           //enable of single controller actions
           //----------------------------------- 
           IF ("AC".CTL_AV_SPD_TI > 0.0)   THEN         //i- part
               #int_action_on   :=  true;
           ELSE
               #int_action_on   :=  false;
           END_IF;

           IF ("AC".CTL_AV_SPD_TD > 0.0)   THEN         //d-part
               #der_action_on   :=  true;
           ELSE
               #der_action_on   :=  false;
           END_IF;

           //call Standard PID controller 
           //----------------------------
           #STD_PID(COM_RST         :=  "KYD".SPD_CTRL_RST,                   //restart of controller, resets controller values
                   MAN_ON          :=  NOT #ctl_avg_spd_on,                 //switch controller on/off
                   PVPER_ON        :=  false,                              //activate reading of peripherie value
                   P_SEL           :=  true,                               //proportional action on
                   I_SEL           :=  #int_action_on,                      //integral action on
                   INT_HOLD        :=  #int_hold_req,                       //integral action hold
                   I_ITL_ON        :=  false,                              //initialization of the integral action - set value of I_ITLVAL
                   D_SEL           :=  #der_action_on,                      //derivative action on
                   CYCLE           :=  T#100ms,                            //sample time
                   SP_INT          :=  #set,                                //internal setpoint
                   PV_IN           :=  #act,                                //process variable input
                   PV_PER          :=  W#16#0000,                          //process variable peripherial input
                   MAN             :=  #hand,                               //hand value as percentaged input
                   GAIN            :=  "AC".CTL_AV_SPD_GN,                   //controller gain
                   TI              :=  DINT_TO_TIME(REAL_TO_DINT("AC".CTL_AV_SPD_TI * 1000.0)),  //integration time
                   TD              :=  DINT_TO_TIME(REAL_TO_DINT("AC".CTL_AV_SPD_TD * 1000.0)),  //derivative time
                   TM_LAG          :=  DINT_TO_TIME(REAL_TO_DINT("AC".CTL_AV_SPD_T1 * 1000.0)),  //time lag of the derivative action
                   DEADB_W         :=  0.0,                            //dead band of control deviation
                   LMN_HLM         :=  #hl,                             //upper limit of controller output as percentaged value 
                   LMN_LLM         :=  #ll,                             //lower limit of controller output as percentaged value
                   PV_FAC          :=  1.0,                            //process variable factor (used on peripherial input)
                   PV_OFF          :=  0.0,                            //process variable offset
                   LMN_FAC         :=  1.0,                            //output standardization(percentage to physical value)
                   LMN_OFF         :=  0.0,                            //offset of output value
                   I_ITLVAL        :=  0.0,                            //initialization value of the integral action
                   DISV            :=  #z_input);                       //disturbance variable

                   //write output variables of PID controller
                   //----------------------------------------
                   "CTL".Y_AVG_XT_SPD    :=  #STD_PID.LMN * #ro;               //controller output variable as physical value

                   #per_out         :=  #STD_PID.LMN_PER;    //peripherial controller output variable
                   #high_lim_active :=  #STD_PID.QLMN_HLM;   //high limit of controller output is reached
                   #low_lim_active  :=  #STD_PID.QLMN_LLM;   //low limit of controller output is reached
                   #p_part_out      :=  #STD_PID.LMN_P;      //proportionality component
                   #i_part_out      :=  #STD_PID.LMN_I;      //integral component
                   #d_part_out      :=  #STD_PID.LMN_D;      //derivative component
                   #eff_act_val     :=  #STD_PID.PV;         //effective process variable 
                   #error_sig       :=  #STD_PID.ER;         //control deviation

           //write display values of controller parts
           //----------------------------------------        
           "DIS".AVG_SPD_CONT_P  := #p_part_out * #ro; 
           "DIS".AVG_SPD_CONT_D  := #d_part_out * #ro;
           "DIS".AVG_SPD_CONT_I  := #i_part_out * #ro;

           //evaluate controller output limits
           //---------------------------------
           IF #high_lim_active XOR #low_lim_active   THEN                //check controller limits
               IF (#ctrl_calls > 50) THEN                                   
                   IF #high_lim_active AND (#i_part_out > 0.0)   THEN 
                       #int_hold_req    :=  true;                       //set integral action on hold
                   ELSIF #low_lim_active AND (#i_part_out < 0.0) THEN 
                       #int_hold_req    :=  true;                       //set integral action on hold
                   ELSE 
                       #int_hold_req    :=  false;                      //reset integral action on hold
                   END_IF;
               ELSE
                   #ctrl_calls  :=  #ctrl_calls + 1;                     //count controller calls
               END_IF;
           ELSE
               #ctrl_calls      :=  0;                                  //reset controller call counts
               #int_hold_req    :=  false;                              //reset integral action hold request
           END_IF;

           //switch on average pull speed controller
           //--------------------------------------- 
           IF "SY".CTL_AVG_SPD_ON    THEN 
               #ctl_avg_spd_on  :=  true;
           END_IF;


       //write average speed controller output as setpoint for crucible rotation
       //-----------------------------------------------------------------------    
       IF ("APC".STATUS = "APC".SHOULDER) AND ("PAR_MAIN".SH_CRUC_ROT_CTL_ON = 1.0) THEN
           "CTL".SET_CR_ROT  :=  "CTL".Y_GRW_RTE;
       ELSIF ("APC".STATUS = "APC".BODY) AND ("PAR_MAIN".BY_CRUC_ROT_CTL_ON = 1.0) THEN    
           "CTL".SET_CR_ROT  :=  "CTL".Y_AVG_XT_SPD;
       END_IF;         

       //save actual values for next cycle
       //---------------------------------               
       #z_input_old             :=  #z_input;
       #set_avg_cruc_rot_old    :=  "AC".SET_AVG_CRUC_ROT;
END_FUNCTION_BLOCK

FUNCTION_BLOCK "CM_LOOP_MLT_TMP"   // FB139, SCL
{ S7_Optimized_Access := 'FALSE' }
VERSION : 0.0
// --------------------------------------------------------------------------------
//     program     :    CM_LOOP_MLT_TMP
//     description :    melt temperature control loop 
//     name        :    K. Kalkowski
//     date        :    10.12.99 
// 
//     revision    :    call of CONT_C added as alternative
//     name        :    G. Eibelsh鋟ser
//     date        :    07.09.2007
//     
//     revision    :    
//     name        :    
//     date        :    
// 
//                     (c)PVA TePla AG
//     --------------------------------------------------------------------------------
   VAR
      STD_PID : CONT_C;   // standard Siemens controller algorithm
      PT1 : "CM_PT1";   // pt1 filter for melt temp
      ramp_enb : Bool;
      cyc_cnt : Bool;
      int_hold_req : Bool;   // integral hold action request
      pyr_failed : Bool;
      ctl_mlt_tmp_on : Bool;
      ctrl_calls : Int;   // controller call counter
      i : Int;
      set : Real;   // internal set point
      act : Real;   // internal actual value
      set_ramp : Real;
      pyr_act_melt_tmp_prv : Real;
      set_prv_cyc : Real;
   END_VAR
   VAR_TEMP
      high_lim_active : Bool;   // high limit of controller output is reached
      low_lim_active : Bool;   // low limit of controller output is reached
      int_action_on : Bool;   // integral action on
      der_action_on : Bool;   // derivative action on
      per_out : Word;   // peripherial controller output variable
      p_part_out : Real;   // proportionality component
      i_part_out : Real;   // integral component
      d_part_out : Real;   // derivative component
      eff_act_val : Real;   // effective process variable
      error_sig : Real;   // control deviation
   END_VAR
   VAR CONSTANT
      nc : Real := 0.0;   // "not connected" input
   END_VAR
BEGIN

       //read setpoint from recipe
       //-------------------------                                                
       #set := "AC".SET_MLT_1_TMP;              

       //read filter time from recipe
       //----------------------------
       "AC".CTL_MLT_TMP_1_TF := "PAR_SUB".FI_MLT_TMP_1;

       //call filter algorithm
       //---------------------                                                  
       #PT1 (u_in      := "PAI".PYR_ACT_MELT_TMP,                   
            t1_in     := "AC".CTL_MLT_TMP_1_TF, 
            ts_in     := 0.1,
            tc_in     := 0.1,
            range_in  := "CNF".MLT_TMP_1_RANGE_HI,
            range_out := "CNF".MLT_TMP_1_RANGE_HI,
            y_llim    := "CNF".MLT_TMP_1_RANGE_LOW,
            y_hlim    := "CNF".MLT_TMP_1_RANGE_HI,
            y_out     := "CTL".AVG_MLT_1_TMP);

       "CTL".AVG_MLT_1_TMP   := "CTL".AVG_MLT_1_TMP + "PAR_MAIN".MCONST_MLT_TMP_OFFS;  //add offset to filtered value                          

       #act                 := "CTL".AVG_MLT_1_TMP;
       (*
       //check pyrometer signal when temperature control is on
       //-----------------------------------------------------
       IF SY.CTL_MLT_TMP_ON  THEN
           //calculate deviation of temperature from last cycle
           //--------------------------------------------------
           IF ((pyr_act_melt_tmp_prv - PAI.PYR_ACT_MELT_TMP) > 15.0) THEN  //temp. drop larger 15癈
               pyr_failed  :=  true;
           END_IF;

       ELSE
           //reset signal "pyrometer failed" with delay
           //------------------------------------------
           IF pyr_failed   THEN 
               IF (i > 50)    THEN             //delay reset at least 5 seconds
                   IF NOT APC.AUTOMATIC THEN
                       pyr_failed  :=  false;  //reset failure flag when automatic is off
                   END_IF;
               ELSE 
                   i   :=  i + 1;  //increment 100ms counter
               END_IF; 
           ELSE 
               i   :=  0;  //reset counter value
           END_IF;

       END_IF; 

       //store actual temperature for one 100ms cycle
       //--------------------------------------------
       pyr_act_melt_tmp_prv   :=  PAI.PYR_ACT_MELT_TMP;    

       //set fault message when pyrometer failed
       //---------------------------------------
       FLT.MLT_TMP_SIG   :=  pyr_failed;
       *)
       //built control on flag
       //---------------------                                                    
       IF "APC".AUTOMATIC AND NOT #pyr_failed THEN                         
           "SY".CTL_MLT_TMP_ON := "DC".CTL_MLT_1_TMP_ON;                 
       ELSE 
           "SY".CTL_MLT_TMP_ON := FALSE; 
       END_IF;

       "LT".CTL_MELT_TMP_1_ON := "SY".CTL_MLT_TMP_ON; 

       //melt temperature controller setpoint ramp
       //-----------------------------------------
       IF "SY".CTL_MLT_TMP_ON  THEN

           IF (#set <> #set_prv_cyc) THEN    //compare setpoint with setpoint of previous cycle
               #ramp_enb := true;           //enable ramp when setpoint has changed
           END_IF;
           #set_prv_cyc :=  #set;        //store setpoint of current cycle

           // call setpoint ramp function after controller start
           //---------------------------------------------------
           IF ("PAR_SUB".MELT_TMP_RP_GRAD > 0.0)     THEN
               "CM_SET_RAMP"(rp_enb      := #ramp_enb,
                           i           := #cyc_cnt,
                           max_dev     := "PAR_SUB".MELT_TMP_RP_MAX_DEV,
                           rp_start    := "PAR_SUB".MELT_TMP_RP_START,
                           rp_grad     := "PAR_SUB".MELT_TMP_RP_GRAD,
                           tme_base    := 60.0,
                           tc_in       := 0.1,
                           set_p       := #set,
                           act_v       := #act,
                           set_out     := #set_ramp);

               #set     := #set_ramp; 
           END_IF;
       ELSE
           #ramp_enb  := true;     
           #cyc_cnt   := true;                
       END_IF;

       //set display variables of melt temperature
       //-----------------------------------------
       "DIS".SET_MLT_TMP_1   := #set;
       "DIS".ACT_MLT_TMP_1   := #act;

       //do controller call
       //------------------ 

           //switch off melt temperature controller
           //-------------------------------------- 
           IF NOT "SY".CTL_MLT_TMP_ON   THEN 
               #ctl_mlt_tmp_on  :=  false;
           END_IF;

           //enable of single controller actions
           //----------------------------------- 
           IF ("AC".CTL_MLT_TMP_1_TI > 0.0)   THEN         //i- part
               #int_action_on   :=  true;
           ELSE
               #int_action_on   :=  false;
           END_IF;

           IF ("AC".CTL_MLT_TMP_1_TD > 0.0)   THEN         //d-part
               #der_action_on   :=  true;
           ELSE
               #der_action_on   :=  false;
           END_IF;

           //call Standard PID controller 
           //----------------------------
           #STD_PID(COM_RST         :=  "KYD".MLT_TMP_CTRL_RST,               //restart of controller, resets controller values
                   MAN_ON          :=  NOT #ctl_mlt_tmp_on,                 //switch controller on/off
                   PVPER_ON        :=  false,                              //activate reading of peripherie value
                   P_SEL           :=  true,                               //proportional action on
                   I_SEL           :=  #int_action_on,                      //integral action on
                   INT_HOLD        :=  #int_hold_req,                       //integral action hold
                   I_ITL_ON        :=  false,                              //initialization of the integral action - set value of I_ITLVAL
                   D_SEL           :=  #der_action_on,                      //derivative action on
                   CYCLE           :=  T#100ms,                            //sample time
                   SP_INT          :=  #set,                                //internal setpoint
                   PV_IN           :=  #act,                                //process variable input
                   PV_PER          :=  W#16#0000,                          //process variable peripherial input
                   MAN             :=  0.0,                                //hand value as percentaged input
                   GAIN            :=  "AC".CTL_MLT_TMP_1_GN,                //controller gain
                   TI              :=  DINT_TO_TIME(REAL_TO_DINT("AC".CTL_MLT_TMP_1_TI * 1000.0)), //integration time
                   TD              :=  DINT_TO_TIME(REAL_TO_DINT("AC".CTL_MLT_TMP_1_TD * 1000.0)), //derivative time
                   TM_LAG          :=  DINT_TO_TIME(REAL_TO_DINT("AC".CTL_MLT_TMP_1_T1 * 1000.0)), //time lag of the derivative action
                   DEADB_W         :=  0.0,                            //dead band of control deviation
                   LMN_HLM         :=  100.0,                          //upper limit of controller output as percentaged value 
                   LMN_LLM         :=  -100.0,                         //lower limit of controller output as percentaged value
                   PV_FAC          :=  1.0,                            //process variable factor (used on peripherial input)
                   PV_OFF          :=  0.0,                            //process variable offset
                   LMN_FAC         :=  1.0,                            //output standardization(percentage to physical value)
                   LMN_OFF         :=  0.0,                            //offset of output value
                   I_ITLVAL        :=  0.0,                            //initialization value of the integral action
                   DISV            :=  #nc);                            //disturbance variable

                   //write output variables of PID controller
                   //----------------------------------------
                   "CTL".Y_MLT_1_TMP :=  #STD_PID.LMN / 100.0 * "CNF".HTR_1_TMP_RANGE_HI;   //controller output variable as physical value

                   #per_out         :=  #STD_PID.LMN_PER;                    //peripherial controller output variable
                   #high_lim_active :=  #STD_PID.QLMN_HLM;                   //high limit of controller output is reached
                   #low_lim_active  :=  #STD_PID.QLMN_LLM;                   //low limit of controller output is reached
                   #p_part_out      :=  #STD_PID.LMN_P;                      //proportionality component
                   #i_part_out      :=  #STD_PID.LMN_I;                      //integral component
                   #d_part_out      :=  #STD_PID.LMN_D;                      //derivative component
                   #eff_act_val     :=  #STD_PID.PV;                         //effective process variable 
                   #error_sig       :=  #STD_PID.ER;                         //control deviation

           //evaluate controller output limits
           //---------------------------------
           IF #high_lim_active XOR #low_lim_active   THEN                //check controller limits
               IF (#ctrl_calls > 50) THEN                                   
                   IF #high_lim_active AND (#i_part_out > 0.0)   THEN 
                       #int_hold_req    :=  true;                       //set integral action on hold
                   ELSIF #low_lim_active AND (#i_part_out < 0.0) THEN 
                       #int_hold_req    :=  true;                       //set integral action on hold
                   ELSE 
                       #int_hold_req    :=  false;                      //reset integral action on hold
                   END_IF;
               ELSE
                   #ctrl_calls  :=  #ctrl_calls + 1;                     //count controller calls
               END_IF;
           ELSE
               #ctrl_calls      :=  0;                                  //reset controller call counts
               #int_hold_req    :=  false;                              //reset integral action hold request
           END_IF;

           //switch on melt temperature controller
           //------------------------------------- 
           IF "SY".CTL_MLT_TMP_ON   THEN 
               #ctl_mlt_tmp_on  :=  true;
           END_IF;
END_FUNCTION_BLOCK

FUNCTION_BLOCK "CM_LOOP_GRW_RTE"   // FB140, SCL
{ S7_Optimized_Access := 'FALSE' }
VERSION : 0.0
// --------------------------------------------------------------------------------
//     program     :    CM_LOOP_GRW_RTE
//     description :    growth rate control loop 
//     name        :    K. Kalkowski
//     date        :    12.12.99
// 
//     revision    :    call of CONT_C added as alternative
//     name        :    G. Eibelsh鋟ser
//     date        :    07.09.2007
//     
//     revision    :    
//     name        :    
//     date        :    
// 
//                     (c)PVA TePla AG
//     --------------------------------------------------------------------------------
   VAR
      STD_PID : CONT_C;   // standard Siemens controller algorithm
      DT1 : "CM_DT1";   // dt1 filter for act gtrowth rate
      ramp_enb : Bool;
      cyc_cnt : Bool;
      int_hold_req : Bool;   // integral hold action request
      ctl_grw_rte_on : Bool;
      ctrl_calls : Int;   // controller call counter
      set : Real;   // internal set point
      act : Real;   // internal actual value
      hand : Real;   // internal hand value
      ll : Real;   // controller output low limit
      hl : Real;   // controller output high limit
      ro : Real;   // controller output range
      set_ramp : Real;
      z_input : Real;   // interference input
      z_input_old : Real;   // interference input of previous cycle
      set_avg_cruc_rot_old : Real;   // average crucible rotation setpoint of previous cycle
   END_VAR
   VAR_TEMP
      high_lim_active : Bool;   // high limit of controller output is reached
      low_lim_active : Bool;   // low limit of controller output is reached
      int_action_on : Bool;   // integral action on
      der_action_on : Bool;   // derivative action on
      per_out : Word;   // peripherial controller output variable
      p_part_out : Real;   // proportionality component
      i_part_out : Real;   // integral component
      d_part_out : Real;   // derivative component
      eff_act_val : Real;   // effective process variable
      error_sig : Real;   // control deviation
      act_tmp : Real;   // internal actual value
   END_VAR
   VAR CONSTANT
      nc : Real := 0.0;   // "not connected" input
   END_VAR
BEGIN


       IF "PAR_MAIN".SH_CRUC_ROT_CTL_ON = 1.0 THEN
           IF   ("APC".STATUS = "APC".SHOULDER)   THEN

               IF  "APC".AUTOMATIC  AND NOT "SY".CTL_CR_ROT_SMI    THEN  
                   IF  "DV".START_SH_FLAG     THEN
                       #hand    :=  "PAR_MAIN".SH_START_CRUC_ROT; //crucible rotation setpoint provided from main page
                   ELSIF "DV".TRANS_SH_BY_FLAG  THEN
                       #hand    := "CTL".SET_CR_ROT;              //keep last controller setpoint as setpoint for transistion    
                   END_IF;           
               ELSE
                   #hand := "CM_INSELECT" (auto  := ("APC".AUTOMATIC AND NOT "SY".CTL_CR_ROT_SMI),        
                                       track  := false,
                                       ac     := "AC".SET_CR_ROT,                
                                       kya    := "KYA".SET_CR_ROT);
               END_IF;

               //transform to percentage value
               //-----------------------------
               IF "DV".GRW_RTE_CTRL_STD_ALG  THEN    //only when standard PID algorithm is active
                   #hand    :=  #hand / "CNF".CR_ROT_RANGE * 100.0;
               END_IF;

           END_IF;
       ELSE
           #hand := 0.0;
       END_IF;   

       //read setpoint from recipe
       //-------------------------                              
       #set := "AC".SET_GRW_RTE;         

       //read filter time from recipe
       //----------------------------
       "AC".CTL_GRO_TF := "PAR_SUB".FI_GRO_SH;                

       //call derivative algorithm
       //-------------------------
       #DT1 (u_in       := "AV".ACT_XT_DIA * 600,                   //build actual value   
            td_in      := 0.10,                //mm/min                                
            t1_in      := "AC".CTL_GRO_TF, 
            ts_in      := 1.0,
            tc_in      := 0.1,
            range_in   := "CNF".XT_LFT_RANGE,  
            range_out  := "CNF".XT_LFT_RANGE,
            y_llim     := ("CNF".XT_LFT_RANGE * (-1)),
            y_hlim     := "CNF".XT_LFT_RANGE,
            y_out      := "CTL".ACT_GRW_RTE);

       "DIS".ACT_XTAL_GRO := "CTL".ACT_GRW_RTE;
       #act              := "CTL".ACT_GRW_RTE;                 

       //build control on flag
       //---------------------
       IF "APC".AUTOMATIC THEN                               
           IF "SY".CTL_AVG_CRUC_ROT_ON   THEN
               IF  NOT "SY".CTL_CR_ROT_SMI   THEN
                   "SY".CTL_GRW_RTE_ON := "DC".CTL_GRW_RTE_ON; //set flag according to process mode                 
               ELSE 
                   "SY".CTL_GRW_RTE_ON := FALSE;             //switch off if cruc rot is in semi mode
               END_IF;
           ELSE    
               IF NOT "SY".CTL_HTR_1_SMI THEN 
                   "SY".CTL_GRW_RTE_ON := "DC".CTL_GRW_RTE_ON; //set flag according to process mode
               ELSE
                   "SY".CTL_GRW_RTE_ON := FALSE;
               END_IF;        
           END_IF;
       ELSE
           "SY".CTL_GRW_RTE_ON := FALSE;                     //switch off growth rate control in manuell mode
       END_IF;        

       "LT".CTL_GRO_ON := "SY".CTL_GRW_RTE_ON;                 //set light variable for growth control on         

       //check controller output range
       //-----------------------------
       IF ("APC".STATUS = "APC".SHOULDER)  AND ("PAR_MAIN".SH_CRUC_ROT_CTL_ON = 1.0)  THEN

           IF "SY".CTL_GRW_RTE_ON    THEN
               IF "DV".GRW_RTE_CTRL_STD_ALG  THEN 
                   #ll  :=  "AC".SET_CRUC_ROT_DEV_2 / "CNF".CR_ROT_RANGE * 100.0;
                   #hl  :=  "AC".SET_CRUC_ROT_DEV_1 / "CNF".CR_ROT_RANGE * 100.0;
                   #ro  :=  "CNF".CR_ROT_RANGE / 100.0;
               ELSE
                   #ll  :=  "AC".SET_CRUC_ROT_DEV_2;
                   #hl  :=  "AC".SET_CRUC_ROT_DEV_1;
                   #ro  :=  "CNF".CR_ROT_RANGE;
               END_IF;

           ELSE
               IF "DV".GRW_RTE_CTRL_STD_ALG  THEN 
                   #ll  :=  0.0;
                   #hl  :=  100.0;
                   #ro  :=  "CNF".CR_ROT_RANGE / 100.0;
               ELSE
                   #ll  :=  0.0;
                   #hl  :=  "CNF".CR_ROT_RANGE;
                   #ro  :=  "CNF".CR_ROT_RANGE;
               END_IF;
           END_IF;      
       ELSE
           IF "DV".GRW_RTE_CTRL_STD_ALG  THEN 
               #ll  :=  -100.0;
               #hl  :=  100.0;
               #ro  :=  "CNF".HTR_1_TMP_RANGE_HI / 100.0;
           ELSE
               #ll  :=  "CNF".HTR_1_TMP_RANGE_HI *(-1);
               #hl  :=  "CNF".HTR_1_TMP_RANGE_HI;
               #ro  :=  "CNF".HTR_1_TMP_RANGE_HI;
           END_IF;
       END_IF;

       IF "SY".CTL_GRW_RTE_ON  THEN
           // call setpoint ramp function after controller start
           //---------------------------------------------------
           IF ("PAR_SUB".GRO_RP_GRAD > 0.0)     THEN
               IF #act < 0.0    THEN
                   #act_tmp := 0.0;     //set act_tmp to zero if act < zero
               ELSE
                   #act_tmp := #act;        
               END_IF;    

               "CM_SET_RAMP"(rp_enb      := #ramp_enb,
                           i           := #cyc_cnt,
                           max_dev     := "PAR_SUB".GRO_RP_MAX_DEV,
                           rp_start    := "PAR_SUB".GRO_RP_START,
                           rp_grad     := "PAR_SUB".GRO_RP_GRAD,
                           tme_base    := 60.0,
                           tc_in       := 0.1,
                           set_p       := #set,
                           act_v       := #act_tmp,
                           set_out     := #set_ramp);

               #set     := #set_ramp; 
           END_IF;
       ELSE
           #ramp_enb  := TRUE;     
           #cyc_cnt   := TRUE;                
       END_IF;
       //write display value with setpoint
       //---------------------------------
       "DIS".SET_XTAL_GRO := #set;

       //reset saved interference variables for cruc rot control if growth rate controller is off
       //----------------------------------------------------------------------------------------
       IF   "SY".CTL_GRW_RTE_ON =   FALSE    THEN
           #z_input_old          := 0.0;
           #set_avg_cruc_rot_old := "AC".SET_AVG_CRUC_ROT;
       END_IF;                            

       //change polarity of setpoint and actual if crucible rotation control is off
       //--------------------------------------------------------------------------
       IF ("PAR_MAIN".SH_CRUC_ROT_CTL_ON = 0.0) THEN
           #set     := #set *(-1);
           #act     := #act *(-1);
           #z_input := 0.0;             // keep interference input 0.0, if crucible rotation control is off

       //set interference input with average crucible rotation profile
       //-----------------------------------------------------------------    
       ELSE
           #z_input := #z_input_old + (#set_avg_cruc_rot_old - "AC".SET_AVG_CRUC_ROT) * (-1);   

           //transform to percentage value when standard algorithm is set
           //------------------------------------------------------------
           IF "DV".GRW_RTE_CTRL_STD_ALG  THEN
               #z_input := #z_input / "CNF".CR_ROT_RANGE * 100.0;
           END_IF;
       END_IF;        

       //do controller call
       //------------------

           //switch off growth rate controller
           //---------------------------------
           IF NOT "SY".CTL_GRW_RTE_ON   THEN 
               #ctl_grw_rte_on  :=  false;
           END_IF;

           //enable of single controller actions
           //----------------------------------- 
           IF ("AC".CTL_GRO_TI > 0.0)   THEN             //i- part
               #int_action_on   :=  true;
           ELSE
               #int_action_on   :=  false;
           END_IF;

           IF ("AC".CTL_GRO_TD > 0.0)   THEN             //d-part
               #der_action_on   :=  true;
           ELSE
               #der_action_on   :=  false;
           END_IF;

           //call Standard PID controller 
           //----------------------------
           #STD_PID(COM_RST         :=  "KYD".GRW_RTE_CTRL_RST,               //restart of controller, resets controller values
                   MAN_ON          :=  NOT #ctl_grw_rte_on,                //switch controller on/off
                   PVPER_ON        :=  false,                              //activate reading of peripherie value
                   P_SEL           :=  true,                               //proportional action on
                   I_SEL           :=  #int_action_on,                      //integral action on
                   INT_HOLD        :=  #int_hold_req,                       //integral action hold
                   I_ITL_ON        :=  false,                              //initialization of the integral action - set value of I_ITLVAL
                   D_SEL           :=  #der_action_on,                      //derivative action on
                   CYCLE           :=  T#100ms,                            //sample time
                   SP_INT          :=  #set,                                //internal setpoint
                   PV_IN           :=  #act,                                //process variable input
                   PV_PER          :=  W#16#0000,                          //process variable peripherial input
                   MAN             :=  #hand,                               //hand value as percentaged input
                   GAIN            :=  "AC".CTL_GRO_GN,                      //controller gain
                   TI              :=  DINT_TO_TIME(REAL_TO_DINT("AC".CTL_GRO_TI * 1000.0)), //integration time
                   TD              :=  DINT_TO_TIME(REAL_TO_DINT("AC".CTL_GRO_TD * 1000.0)), //derivative time
                   TM_LAG          :=  DINT_TO_TIME(REAL_TO_DINT("AC".CTL_GRO_T1 * 1000.0)), //time lag of the derivative action
                   DEADB_W         :=  0.0,                            //dead band of control deviation
                   LMN_HLM         :=  #hl,                             //upper limit of controller output as percentaged value 
                   LMN_LLM         :=  #ll,                             //lower limit of controller output as percentaged value
                   PV_FAC          :=  1.0,                            //process variable factor (used on peripherial input)
                   PV_OFF          :=  0.0,                            //process variable offset
                   LMN_FAC         :=  1.0,                            //output standardization(percentage to physical value)
                   LMN_OFF         :=  0.0,                            //offset of output value
                   I_ITLVAL        :=  0.0,                            //initialization value of the integral action
                   DISV            :=  #z_input);                       //disturbance variable

                   //write output variables of PID controller
                   //----------------------------------------
                   "CTL".Y_GRW_RTE   :=  #STD_PID.LMN * #ro;                   //controller output variable as physical value

                   #per_out         :=  #STD_PID.LMN_PER;                    //peripherial controller output variable
                   #high_lim_active :=  #STD_PID.QLMN_HLM;                   //high limit of controller output is reached
                   #low_lim_active  :=  #STD_PID.QLMN_LLM;                   //low limit of controller output is reached
                   #p_part_out      :=  #STD_PID.LMN_P;                      //proportionality component
                   #i_part_out      :=  #STD_PID.LMN_I;                      //integral component
                   #d_part_out      :=  #STD_PID.LMN_D;                      //derivative component
                   #eff_act_val     :=  #STD_PID.PV;                         //effective process variable 
                   #error_sig       :=  #STD_PID.ER;                         //control deviation

           //write display values of controller parts
           //----------------------------------------        
           "DIS".GRW_RTE_CONT_P:= #p_part_out * #ro; 
           "DIS".GRW_RTE_CONT_I:= #i_part_out * #ro;
           "DIS".GRW_RTE_CONT_D:= #d_part_out * #ro;

           //evaluate controller output limits
           //---------------------------------
           IF #high_lim_active XOR #low_lim_active   THEN                //check controller limits
               IF (#ctrl_calls > 50) THEN                                   
                   IF #high_lim_active AND (#i_part_out > 0.0)   THEN 
                       #int_hold_req    :=  true;                       //set integral action on hold
                   ELSIF #low_lim_active AND (#i_part_out < 0.0) THEN 
                       #int_hold_req    :=  true;                       //set integral action on hold
                   ELSE 
                       #int_hold_req    :=  false;                      //reset integral action on hold
                   END_IF;
               ELSE
                   #ctrl_calls  :=  #ctrl_calls + 1;                     //count controller calls
               END_IF;
           ELSE
               #ctrl_calls      :=  0;                                  //reset controller call counts
               #int_hold_req    :=  false;                              //reset integral action hold request
           END_IF;

           //switch on growth rate controller
           //--------------------------------
           IF "SY".CTL_GRW_RTE_ON   THEN 
               #ctl_grw_rte_on  :=  true;
           END_IF;

       //save actual values for next cycle
       //---------------------------------               
       #z_input_old             :=  #z_input;
       #set_avg_cruc_rot_old    :=  "AC".SET_AVG_CRUC_ROT;
END_FUNCTION_BLOCK

FUNCTION_BLOCK "CM_LOOP_MLT_LVL"   // FB141, SCL
{ S7_Optimized_Access := 'FALSE' }
VERSION : 0.0
// --------------------------------------------------------------------------------
//     program     :    CM_LOOP_MLT_LVL
//     description :    melt level control loop 
//     name        :    K. Kalkowski
//     date        :    08.12.99 
// 
//     revision    :    
//     name        :    
//     date        :    
// 
//                     (c)PVA TePla AG
//     --------------------------------------------------------------------------------
   VAR
      P : "CM_P";   // p controller melt level
      PT1 : "CM_PT1";   // pt1 filter for melt level
      ramp_enb : Bool;
      cyc_cnt : Bool;
      enb_mlt_lvl_sft : Bool;
      set : Real;   // internal set point
      act : Real;   // internal actual value
      hand : Real;   // internal hand value
      set_ramp : Real;
      set_cr_spd_cof : Real;
      mlt_lvl_sft_dur : Real;
      act_mlt_lvl_sft : Real;
      mlt_lvl_sft_len : Real;
      mlt_lvl_sft_str_len : Real;
      mlt_lvl_sft_offs_spd : Real;
   END_VAR
   VAR CONSTANT
      nc : Real := 0.0;   // "not connected" input
      min_cr_spd : Real := 0.001;   // [mm/min]
      min_lvl_sft_len : Real := 0.1;   // [mm]
      safety_gap : Real := 5.0;   // safety gap melt level - funnel in [mm]
   END_VAR
BEGIN

       //build hand value 
       //----------------
       IF ("CTL".SET_SPEED_OFFS = 0.0) THEN  //offset speed controller off and output ramped down to zero 
           #hand := "CM_INSELECT" (auto   := ("APC".AUTOMATIC AND NOT "SY".CTL_MLT_LVL_SMI),  //hand value used when melt level controller is off       
                                track  := false,
                                ac     := "AC".SET_CR_SPD,                
                                kya    := "KYA".SET_CR_SPD);  
       ELSE
           #hand := "CTL".SET_CR_SPD; //keep melt level controller output as hand value as long as output of offset speed controller is ramp down to zero
       END_IF;

      //crucible speed coeffizient while tracing of pulling speed is active
      //------------------------------------------------------------------- 
      #set_cr_spd_cof := "CM_INSELECT"   (auto   := ("APC".AUTOMATIC AND NOT "SY".CTL_CR_SPD_COF_SMI),        
                                       track  := true,
                                       ac     := "AC".SET_CR_SPD_COF,                
                                       kya    := "KYA".SET_CR_SPD_COF);                      

       //read filter time from recipe
       //----------------------------
       "AC".CTL_MLT_LVL_TF := "PAR_SUB".FI_MLT_LVL;    

       //built control on flag
       //----------------------
       IF "APC".AUTOMATIC AND NOT "SY".CTL_MLT_LVL_SMI THEN
           "SY".CTL_MLT_LVL_ON := "DC".CTL_MLT_LVL_ON;                 
       ELSE 
           "SY".CTL_MLT_LVL_ON := FALSE; 
       END_IF;

       IF "SY".CTL_MLT_LVL_ON  THEN
           // call setpoint ramp function after controller start
           //---------------------------------------------------
           IF ("PAR_SUB".MLT_LVL_RP_GRAD > 0.0)     THEN

               "CM_SET_RAMP"(rp_enb      := #ramp_enb,
                           i           := #cyc_cnt,
                           max_dev     := "PAR_SUB".MLT_LVL_RP_MAX_DEV,
                           rp_start    := "PAR_SUB".MLT_LVL_RP_START,
                           rp_grad     := "PAR_SUB".MLT_LVL_RP_GRAD,
                           tme_base    := 60.0,
                           tc_in       := 0.1,
                           set_p       := #set,
                           act_v       := #act,
                           set_out     := #set_ramp);

               #set     := #set_ramp; 
           END_IF;
       ELSE
           #ramp_enb  := TRUE;     
           #cyc_cnt   := TRUE;                
       END_IF;


       "LT".CTL_LVL_ON := "SY".CTL_MLT_LVL_ON;                             

       //call P controller
       //-----------------
       #P (set_in        := #set,                        
          act_in        := #act,                
          z_in          := "AV".CRUC_RATIO * "CTL".AVG_XT_SPD * ((#set_cr_spd_cof + "CTL".SET_CR_SPD_COF_OFFS) / 100.0),               
          p_in          := "AC".CTL_MLT_LVL_GN,             
          ts_in         := 0.1,                
          tc_in         := 0.1,            
          tw_in         := 0.5,                
          hand_in       := #hand,            
          range_in      := "CNF".LSR_LVL_RANGE,           //100,               
          range_out     := "CNF".CR_LFT_RANGE,             
          y_llim        := 0.0,                         //(CNF.CR_LFT_RANGE *(-1)),              
          y_hlim        := "CNF".CR_LFT_RANGE,         
          ctrl_on       := "SY".CTL_MLT_LVL_ON,               
          hand_lim_dis  := ("APC".AUTOMATIC AND "DC".CR_LFT_FST),              
          y_out         := "CTL".SET_CR_SPD);         

       //write display value
       //-------------------
       "DIS".SET_CR_SPD_COF  :=  #set_cr_spd_cof;     //write recipe value of crucible speed coefficient to display value

       //set enable flag for melt level shift
       //------------------------------------
       IF ("APC".STATUS = "APC".BODY) THEN
          #mlt_lvl_sft_len       := "PAR_MAIN".BY_MLT_LVL_SFT_LEN;
          #mlt_lvl_sft_str_len   := "PAR_MAIN".BY_MLT_LVL_SFT_STR_LEN;
          #mlt_lvl_sft_offs_spd  := "PAR_MAIN".BY_MLT_LVL_SFT_OFFS_SPD;
       ELSE
          #mlt_lvl_sft_len       := "PAR_MAIN".SH_MLT_LVL_SFT_LEN;
          #mlt_lvl_sft_str_len   := "PAR_MAIN".SH_MLT_LVL_SFT_STR_LEN;
          #mlt_lvl_sft_offs_spd  := "PAR_MAIN".SH_MLT_LVL_SFT_OFFS_SPD;
       END_IF;    

       IF ((ABS(#mlt_lvl_sft_len) < #min_lvl_sft_len) OR (#mlt_lvl_sft_offs_spd < #min_cr_spd)) THEN
           #enb_mlt_lvl_sft     :=  false;
           "FLT".SH_MLT_LVL_SFT  :=  FALSE;
       //negative melt level shift length means lift up of melt level and reduction of melt gap
       //--------------------------------------------------------------------------------------
       ELSIF (("PAR_MAIN".ME_GAP_MLT_FNL > #safety_gap) AND ((#mlt_lvl_sft_len * (-1)) < ("PAR_MAIN".ME_GAP_MLT_FNL - #safety_gap))) THEN 
           #enb_mlt_lvl_sft     :=  true;
           "FLT".SH_MLT_LVL_SFT  :=  FALSE;
       ELSE
           #enb_mlt_lvl_sft :=  false;
           IF ("STA".ACT_STATE = "APC".STATE_RUN) THEN
               "FLT".SH_MLT_LVL_SFT  :=  TRUE;
           ELSE
               "FLT".SH_MLT_LVL_SFT  :=  FALSE;
           END_IF;
       END_IF;

       //melt level shift offset speed calculation in shoulder phase
       //-----------------------------------------------------------
       IF (("APC".STATUS = "APC".BODY) AND "DC".CTL_DIA_ON) OR ("APC".STATUS = "APC".SHOULDER)THEN     //body phase step 400
           IF #enb_mlt_lvl_sft THEN          

               //calculate actual melt level shift
               //---------------------------------
               #act_mlt_lvl_sft := #act_mlt_lvl_sft + ABS("AV".MLT_LVL_SFT_OFFS_SPD) * 0.1 / 60;

               //actual shoulder length reached trigger length
               //---------------------------------------------
               IF ("AV".ACT_XT_LEN >= #mlt_lvl_sft_str_len) THEN
                   //crucible lift is active in automatic mode
                   //-----------------------------------------
                   IF "APC".AUTOMATIC THEN
                       //set speed for melt level shift upwards or downwards
                       //---------------------------------------------------
                       IF (#act_mlt_lvl_sft < ABS(#mlt_lvl_sft_len)) THEN 
                           //reduce gap - increase speed
                           //---------------------------
                           IF ((#mlt_lvl_sft_len < 0.0) OR ("APC".STATUS = "APC".SHOULDER)) THEN    //in shoulder only reduction of gap - increase of melt level and speed - no downwards movement!!! 
                               "AV".MLT_LVL_SFT_OFFS_SPD  := #mlt_lvl_sft_offs_spd;           //add positive speed offset
                           //increase gap - decrease speed
                           //-----------------------------
                           ELSE
                               "AV".MLT_LVL_SFT_OFFS_SPD  := #mlt_lvl_sft_offs_spd * (-1.0);  //add negative speed offset
                           END_IF;
                       ELSE
                           "AV".MLT_LVL_SFT_OFFS_SPD  := 0.0;
                       END_IF;
                   ELSE
                       "AV".MLT_LVL_SFT_OFFS_SPD :=  0.0;
                   END_IF;
               ELSE 
                   "AV".MLT_LVL_SFT_OFFS_SPD :=  0.0;
                   #act_mlt_lvl_sft         :=  0.0;        //reset actual shift length at phase shift
               END_IF;
           ELSE
               "AV".MLT_LVL_SFT_OFFS_SPD :=  0.0;
           END_IF;
       //reset offset speed and actual shift in all other phases
       //-------------------------------------------------------
       ELSE
           "AV".MLT_LVL_SFT_OFFS_SPD :=  0.0;
           #act_mlt_lvl_sft         :=  0.0;
       END_IF;

       //set light flag when shoulder melt level shift is active
       //-------------------------------------------------------
       "LT".SH_MLT_LVL_SFT_RUN   :=  (ABS("AV".MLT_LVL_SFT_OFFS_SPD) >= #min_cr_spd);
END_FUNCTION_BLOCK

FUNCTION_BLOCK "CM_P"   // FB142, SCL
{ S7_Optimized_Access := 'FALSE' }
VERSION : 0.0
// --------------------------------------------------------------------------------
//     program     :    CM_P
//     description :    p controller (melt level control)  
//     name        :    K. Kalkowski
//     date        :    14.12.99
// 
//     revision    :    
//     name        :   
//     date        :   
// 
//                     (c)LEYBOLD SYSTEMS
//     --------------------------------------------------------------------------------
   VAR_INPUT
      set_in : Real;   // set point input
      act_in : Real;   // actual value input
      z_in : Real;   // interference input
      p_in : Real;   // controller gain input
      ts_in : Real;   // controller sample time
      tc_in : Real;   // interrupt time for controller module call (ts/tc>=1, ts/tc=integer!)
      tw_in : Real;   // wait time after ctrl_on (tw/tc>=1, tw/tc=integer!)
      hand_in : Real;   // hand value input
      range_in : Real;   // value for 100% input (e.g. 8mm/min = 100%) used for set_in, act_in
      range_out : Real;   // value for 100% output (e.g. 700C = 100%) used for y_out, hand_in
      y_llim : Real;   // low limit for y_out
      y_hlim : Real;   // high limit for y_out
      ctrl_on : Bool;   // controller on/off (1=on 0=off)
      hand_lim_dis : Bool;   // hlim and llim are active on hand input (0=limit active 1=limit inactive)
   END_VAR
   VAR_IN_OUT
      y_out : Real;   // inc function output
   END_VAR
   VAR
      set : Real;   // set point input
      act : Real;   // actual value input
      y : Real;   // controller output
      z : Real;   // interference
      xd : Real;   // set - act
      y_old : Real;   // previous value of pid components
      ctrl_call_cycle : Int;   // pid algorithm call every (ts/tc) cycles
      ctrl_on_delay : Int;   // wait cycles until p controler becomes active
      hlim_active : Bool;   // hlim active
      llim_active : Bool;   // llim active
   END_VAR
BEGIN

       #set := #set_in / #range_in;                                                      //convert input
       #act := #act_in / #range_in;
       #z   := #z_in / #range_out;
       #xd := #set - #act;                                                               //calculate controller input values

       IF #ctrl_on_delay <= REAL_TO_INT(#tw_in/#tc_in)THEN                               //CTRL ON DELAY 
           #ctrl_on_delay := #ctrl_on_delay + 1;
       END_IF;

       IF #ctrl_on = true THEN                                                         //CTRL ON
           IF  #ctrl_call_cycle >= REAL_TO_INT(#ts_in/#tc_in)THEN                        //wait for next controller call                               
               #ctrl_call_cycle := 1;
               IF #ctrl_on_delay > REAL_TO_INT(#tw_in/#tc_in) THEN                               
                   #y := #xd * #p_in + #z; 
               END_IF; 
           ELSE
               #ctrl_call_cycle := #ctrl_call_cycle + 1;
           END_IF;
       ELSE                                                                           //CTRL OFF
           #ctrl_on_delay := 0;                                                        //reset controller on delay counter
           #ctrl_call_cycle := 1;                                                      //reset controller call cycle counter
           #y := #hand_in / #range_out;                                                  //set output value (ctrl off)
       END_IF;

       IF #y > #y_hlim / #range_out THEN                                                 //limit and convert output                                                                        
           #y := #y_hlim / #range_out;
           #hlim_active := true;
       ELSE
           #hlim_active := false;                                                       
       END_IF;
       IF #y < #y_llim / #range_out THEN
           #y := #y_llim / #range_out;
           #llim_active := true;     
       ELSE
           #llim_active := false;
       END_IF;                                                              

       IF NOT #hand_lim_dis OR #ctrl_on THEN                                            //hand limit disable                                                          
           #y_out := #y * #range_out;
       ELSE
           #y_out := #hand_in; 
       END_IF;
END_FUNCTION_BLOCK

FUNCTION_BLOCK "CM_LOOP_AVG_CRUC_ROT"   // FB143, SCL
{ S7_Optimized_Access := 'FALSE' }
VERSION : 0.0
// --------------------------------------------------------------------------------
//     program     :    CM_LOOP_AVG_CRUC_ROT
//     description :    average crucible rotation control loop 
//     name        :    G. Eibelsh鋟ser
//     date        :    09.01.2001
// 
//     revision    :    call of CONT_C added as alternative
//     name        :    G. Eibelsh鋟ser
//     date        :    07.09.2007
//     
//     revision    :    
//     name        :    
//     date        :    
// 
//                     (c)PVA TePla AG
//     --------------------------------------------------------------------------------
   VAR
      STD_PID : CONT_C;   // standard Siemens controller algorithm
      PT1 : "CM_PT1";   // pt1 filter for average crucible rotation
      ramp_enb : Bool;
      cyc_cnt : Bool;
      int_hold_req : Bool;   // integral hold action request
      ctl_avg_cruc_rot_on : Bool;
      ctrl_calls : Int;   // controller call counter
      set : Real;   // internal set point
      act : Real;   // internal actual value
      set_ramp : Real;
   END_VAR
   VAR_TEMP
      high_lim_active : Bool;   // high limit of controller output is reached
      low_lim_active : Bool;   // low limit of controller output is reached
      int_action_on : Bool;   // integral action on
      der_action_on : Bool;   // derivative action on
      per_out : Word;   // peripherial controller output variable
      p_part_out : Real;   // proportionality component
      i_part_out : Real;   // integral component
      d_part_out : Real;   // derivative component
      eff_act_val : Real;   // effective process variable
      error_sig : Real;   // control deviation
   END_VAR
   VAR CONSTANT
      nc : Real := 0.0;   // "not connected" input
   END_VAR
BEGIN

       //read setpoint from recipe
       //-------------------------
       #set := "AC".SET_AVG_CRUC_ROT;      

       //read filter time from recipe
       //----------------------------
       IF "APC".STATUS = "APC".SHOULDER THEN 
           "AC".CTL_AV_CRUC_ROT_TF := "PAR_SUB".FI_SH_AV_CRUC_ROT;                
       ELSE
           "AC".CTL_AV_CRUC_ROT_TF := "PAR_SUB".FI_BY_AV_CRUC_ROT;
       END_IF;    

       //call filter algorithm
       //---------------------   
       #PT1 (u_in      := "KYA".SET_CR_ROT,                
            t1_in     := "AC".CTL_AV_CRUC_ROT_TF, 
            ts_in     := 0.1,
            tc_in     := 0.1,
            range_in  := "CNF".CR_ROT_RANGE,
            range_out := "CNF".CR_ROT_RANGE,
            y_llim    := 0.0,
            y_hlim    := "CNF".CR_ROT_RANGE,
            y_out     := "CTL".AVG_CRUC_ROT); 

       "DIS".ACT_AVG_CRUC_ROT := "CTL".AVG_CRUC_ROT;
       #act                  := "CTL".AVG_CRUC_ROT;                                               

       //built control on flag
       //---------------------
       IF "APC".AUTOMATIC THEN    
           "SY".CTL_AVG_CRUC_ROT_ON := "DC".CTL_CRUC_ROT_ON;                 
       ELSE 
           "SY".CTL_AVG_CRUC_ROT_ON := FALSE; 
       END_IF;

       "LT".CTL_AV_CRUC_ROT_ON := "SY".CTL_AVG_CRUC_ROT_ON;            

       IF "SY".CTL_AVG_CRUC_ROT_ON  THEN
           // call setpoint ramp function after controller start
           //---------------------------------------------------
           IF ("PAR_SUB".AV_CRUC_ROT_RP_GRAD > 0.0)     THEN
               "CM_SET_RAMP"(rp_enb      := #ramp_enb,
                           i           := #cyc_cnt,
                           max_dev     := "PAR_SUB".AV_CRUC_ROT_RP_MAX_DEV,
                           rp_start    := "PAR_SUB".AV_CRUC_ROT_RP_START,
                           rp_grad     := "PAR_SUB".AV_CRUC_ROT_RP_GRAD,
                           tme_base    := 60.0,
                           tc_in       := 0.1,
                           set_p       := #set,
                           act_v       := #act,
                           set_out     := #set_ramp);

               #set     := #set_ramp; 
           END_IF;
       ELSE
           #ramp_enb  := TRUE;     
           #cyc_cnt   := TRUE;                
       END_IF;

       //write display value of setpoint value
       //-------------------------------------
       "DIS".SET_AVG_CRUC_ROT := #set;

       //do controller call
       //------------------

           //switch off average crucible rotation controller
           //----------------------------------------------- 
           IF NOT "SY".CTL_AVG_CRUC_ROT_ON   THEN 
               #ctl_avg_cruc_rot_on  :=  false;
           END_IF;

           //enable of single controller actions
           //----------------------------------- 
           IF ("AC".CTL_AV_CRUC_ROT_TI > 0.0)   THEN         //i- part
               #int_action_on   :=  true;
           ELSE
               #int_action_on   :=  false;
           END_IF;

           IF ("AC".CTL_AV_CRUC_ROT_TD > 0.0)   THEN         //d-part
               #der_action_on   :=  true;
           ELSE
               #der_action_on   :=  false;
           END_IF;

           //call Standard PID controller 
           //----------------------------
           #STD_PID(COM_RST         :=  "KYD".CRUC_ROT_CTRL_RST,              //restart of controller, resets controller values
                   MAN_ON          :=  NOT #ctl_avg_cruc_rot_on,            //switch controller on/off
                   PVPER_ON        :=  false,                              //activate reading of peripherie value
                   P_SEL           :=  true,                               //proportional action on
                   I_SEL           :=  #int_action_on,                      //integral action on
                   INT_HOLD        :=  #int_hold_req,                       //integral action hold
                   I_ITL_ON        :=  false,                              //initialization of the integral action - set value of I_ITLVAL
                   D_SEL           :=  #der_action_on,                      //derivative action on
                   CYCLE           :=  T#100ms,                            //sample time
                   SP_INT          :=  #set,                                //internal setpoint
                   PV_IN           :=  #act,                                //process variable input
                   PV_PER          :=  W#16#0000,                          //process variable peripherial input
                   MAN             :=  0.0,                                //hand value as percentaged input
                   GAIN            :=  "AC".CTL_AV_CRUC_ROT_GN,              //controller gain
                   TI              :=  DINT_TO_TIME(REAL_TO_DINT("AC".CTL_AV_CRUC_ROT_TI * 1000.0)), //integration time
                   TD              :=  DINT_TO_TIME(REAL_TO_DINT("AC".CTL_AV_CRUC_ROT_TD * 1000.0)), //derivative time
                   TM_LAG          :=  DINT_TO_TIME(REAL_TO_DINT("AC".CTL_AV_CRUC_ROT_T1 * 1000.0)), //time lag of the derivative action
                   DEADB_W         :=  0.0,                            //dead band of control deviation
                   LMN_HLM         :=  100.0,                          //upper limit of controller output as percentaged value 
                   LMN_LLM         :=  -100.0,                         //lower limit of controller output as percentaged value
                   PV_FAC          :=  1.0,                            //process variable factor (used on peripherial input)
                   PV_OFF          :=  0.0,                            //process variable offset
                   LMN_FAC         :=  1.0,                            //output standardization(percentage to physical value)
                   LMN_OFF         :=  0.0,                            //offset of output value
                   I_ITLVAL        :=  0.0,                            //initialization value of the integral action
                   DISV            :=  #nc);                            //disturbance variable

                   //write output variables of PID controller
                   //----------------------------------------
                   "CTL".Y_AVG_CRUC_ROT  :=  #STD_PID.LMN / 100.0 * "CNF".HTR_1_TMP_RANGE_HI;   //controller output variable as physical value

                   #per_out         :=  #STD_PID.LMN_PER;                    //peripherial controller output variable
                   #high_lim_active :=  #STD_PID.QLMN_HLM;                   //high limit of controller output is reached
                   #low_lim_active  :=  #STD_PID.QLMN_LLM;                   //low limit of controller output is reached
                   #p_part_out      :=  #STD_PID.LMN_P;                      //proportionality component
                   #i_part_out      :=  #STD_PID.LMN_I;                      //integral component
                   #d_part_out      :=  #STD_PID.LMN_D;                      //derivative component
                   #eff_act_val     :=  #STD_PID.PV;                         //effective process variable 
                   #error_sig       :=  #STD_PID.ER;                         //control deviation

           //evaluate controller output limits
           //---------------------------------
           IF #high_lim_active XOR #low_lim_active   THEN                //check controller limits
               IF (#ctrl_calls > 50) THEN                                   
                   IF #high_lim_active AND (#i_part_out > 0.0)   THEN 
                       #int_hold_req    :=  true;                       //set integral action on hold
                   ELSIF #low_lim_active AND (#i_part_out < 0.0) THEN 
                       #int_hold_req    :=  true;                       //set integral action on hold
                   ELSE 
                       #int_hold_req    :=  false;                      //reset integral action on hold
                   END_IF;
               ELSE
                   #ctrl_calls  :=  #ctrl_calls + 1;                     //count controller calls
               END_IF;
           ELSE
               #ctrl_calls      :=  0;                                  //reset controller call counts
               #int_hold_req    :=  false;                              //reset integral action hold request
           END_IF;

           //switch on average crucible rotation controller
           //---------------------------------------------- 
           IF "SY".CTL_AVG_CRUC_ROT_ON   THEN 
               #ctl_avg_cruc_rot_on  :=  true;
           END_IF;
END_FUNCTION_BLOCK

FUNCTION_BLOCK "CM_DYN_WIN"   // FB144, SCL
{ S7_Optimized_Access := 'FALSE' }
VERSION : 0.0
// ------------------------------------------------------------------------------------
//     program     :    CM_DYN_WIN
//     description :    Filter algorithem that dynamically adapts a filter window according
//                      to the inputs around the filter inputs 
//     
//     name        :    G. Eibelsh鋟ser
//     date        :    26.02.2001 (helau)
//     
//                      RR := rejection ratio
//                      RR := amount of valid data inputs / amout of values per second (10) 
// 
//     revision    :    
//     name        :   
//     date        :   
// 
//                     (c)CGS
//     ------------------------------------------------------------------------------------
   VAR_INPUT
      enb : Bool;   // enable signal for filter funtion
      u_in : Real;   // filter input, diameter
      t1_in : Real;   // filter time in sec.
      ts_in : Real;   // filter sample time
      max_delta : Real;
      min_delta : Real;
      rr : Real;
      tc_in : Real;   // interrupt time for filter module call (ts/tc>=1, ts/tc=integer!)
      range_in : Real;   // value for 100% input (e.g. 8mm/min = 100%) used for u_in
      range_out : Real;   // value for 100% output (e.g. 700C = 100%) used for y_out
      y_llim : Real;   // low limit for y_out
      y_hlim : Real;   // high limit for y_out
   END_VAR
   VAR_IN_OUT
      delta : Real;   // valid window increment
      u_avg : Real;   // filter output 1 second old
      y_out : Real;   // average of summed filter inputs
      i_cycle : Int;   // counter variable for filter cycles
      i_count : Int;   // amount of summed filter inputs
   END_VAR
   VAR
      u : Real;   // scaled filter input
      u_sum : Real;   // sum of scaled filter inputs
      d : Real;   // scaled increment for valid window
      hlim_active : Bool;   // hlim active
      llim_active : Bool;   // llim active
      filter_off : Bool;   // filter function off (T1 = 0)
      ctrl_call_cycle : Int;   // filter algorithm call every (ts/tc) cycles
      filter_call_cycle : Int;   // filter algorithm call every (ts/tc) cycles
      d_min : Real;   // min. value for scaled increment
      d_max : Real;   // max. value for scaled increment
      t1_tmp : Real;   // temporary integration time
   END_VAR
   VAR_TEMP
      rate : Real;
      t1_int : Real;   // internal integration time
      rr_int : Real;   // internal reject ratio
   END_VAR
BEGIN


       IF #range_in = 0 THEN                                            //check range_in value
           #u:= 0;
           #d:= 0;
       ELSE
           #u:=     #u_in / #range_in;
           #d:=     #delta / #range_in;
           #d_min:= #min_delta / #range_in;
           #d_max:= #max_delta / #range_in;
       END_IF;

       IF  #ctrl_call_cycle >= REAL_TO_INT(#ts_in/#tc_in)THEN             //wait for next controller call                               
           #ctrl_call_cycle := 1;

           IF #t1_in <= 0.0 OR NOT #enb  THEN
               #filter_off := true;      
           ELSE
               #filter_off := false;      
           END_IF;

           IF #filter_off = false  THEN

               #i_cycle := #i_cycle + 1;     // cycle counter for filter


               //call ramp function to ramp filter time from 0 to recipe value
               //-------------------------------------------------------------
               "CM_RAMP"(u           := #t1_in,                  //input     
                       slope       := 1.0,                    //slope per sec 
                       tc_in       := 0.1,                    //interrupt time for function call 
                       enable      := true,                   //enable ramp function
                       y           := #t1_tmp);                //ramp function output

               //check if reject ratio is > 0
               //----------------------------   
               IF #rr > 0.0 THEN
                   #rr_int := #rr;
               ELSE
                   #rr_int  := 5.0;        // reject ratio = 50 % (default value if no parameter input)
               END_IF;             

               #rate    := #rr_int / 5;   // calculate rate for increment or reduction of window        

               //check if input is inside the valid window
               //-----------------------------------------  
               IF (#u > #u_avg - #d) AND (#u < #u_avg + #d) THEN     //compare actual input with last average input
                   #u_sum   := #u_sum + #u;       //sum input values
                   #i_count := #i_count +1;      //count sum of increments
               END_IF;
               //calculate average input every second
               //------------------------------------
               IF #i_cycle = 10 THEN
                   IF #i_count > 0  THEN
                       #u_avg := #u_sum / #i_count;           //calculate 1 second average of summed filter inputs
                   END_IF;
                   //compare amount of valid data inputs with rejection ratio parameter and adjust window size
                   //-----------------------------------------------------------------------------------------
                   IF #i_count > REAL_TO_INT(#rr_int) THEN 
                       #t1_int  := #t1_tmp * #rate;           //calculate internal integration time
                       #d :=    #d * (1 - #ts_in/#t1_int);     //decrease valid window
                   END_IF;
                   IF #i_count < REAL_TO_INT(#rr_int) THEN
                       #t1_int  := #t1_tmp / #rate;           //calculate internal integration time
                       #d :=    #d / (1 - (#ts_in/#t1_int));   //increase valid window
                   END_IF;  

                   IF #d < #d_min    THEN                    //check minimum value for window
                       #d := #d_min;                         //set minimum value
                   ELSIF #d > 1.0   THEN
                       #d:= 1.0;                            //set maximum value    
                   END_IF;
                   #i_cycle := 0;                           //reset cycle counter
                   #i_count := 0;                           //reset sum counter
                   #u_sum   := 0.0;                         //reset sum variable
               END_IF;    
           ELSE
               //filter is off
               //-------------
               #u_avg               := #u;        //use actual input as average input if filter is off
               #u_sum               := 0.0;      //reset u_sum
               #i_cycle             := 0;        //reset cycle counter
               #i_count             := 0;        //reset value counter
               #d                   := #d_max;    //set start value for delta after filter activation
               #t1_tmp              := 0.0;      //reset integration time
           END_IF;
       ELSE    
           #ctrl_call_cycle := #ctrl_call_cycle + 1;
       END_IF;

       IF #u_avg > #y_hlim / #range_out THEN                              //limit and convert output
           #u_avg := #y_hlim / #range_out;
           #hlim_active := true;
       ELSE
           #hlim_active := false;
       END_IF;
       IF #u_avg < #y_llim / #range_out THEN
           #u_avg := #y_llim / #range_out;
           #llim_active := true;     
       ELSE
           #llim_active := false;
       END_IF;                                                              
       #y_out := #u_avg * #range_out;                                     //set output value   
       #delta := #d * #range_out;                                         //set delta in mm
END_FUNCTION_BLOCK

FUNCTION_BLOCK "CM_LOOP_GAP"   // FB145, SCL
{ S7_Optimized_Access := 'FALSE' }
VERSION : 0.0
// --------------------------------------------------------------------------------
//     program     :    CM_LOOP_GAP
//     description :    gap controller
//     name        :    G. Eibelsh鋟ser
//     date        :    25.08.2020
// 
//     revision    :    
//     name        :    
//     date        :    
// 
//                     (c)PVA TePla AG
//     --------------------------------------------------------------------------------
   VAR
      GAP_PID : CONT_C;   // standard Siemens controller algorithm for Gap Control
      OFFS_SPEED_PID : CONT_C;   // standard Siemens controller algorithm for Speed Control
      int_hold_req_gap : Bool;
      ctl_gap_on : Bool;
      int_hold_req_speed : Bool;
      ctl_offs_spd_on : Bool;
      ctrl_calls_gap : Int;
      ctrl_calls_speed : Int;
      hand_gap : Real;
      hand_offs_spd : Real;
   END_VAR
   VAR_TEMP
      high_lim_active_gap : Bool;   // gap high limit of controller output is reached
      low_lim_active_gap : Bool;   // gap low limit of controller output is reached
      int_action_on_gap : Bool;   // integral action on
      der_action_on_gap : Bool;   // derivative action on
      per_out_gap : Word;   // gap peripherial controller output variable
      p_part_out_gap : Real;   // gap proportionality component
      i_part_out_gap : Real;   // gap integral component
      d_part_out_gap : Real;   // gap derivative component
      eff_act_val_gap : Real;   // gap effective process variable
      error_sig_gap : Real;   // gap control deviation
      high_lim_active_speed : Bool;   // gap high limit of controller output is reached
      low_lim_active_speed : Bool;   // gap low limit of controller output is reached
      int_action_on_speed : Bool;   // integral action on
      der_action_on_speed : Bool;   // derivative action on
      per_out_speed : Word;   // gap peripherial controller output variable
      p_part_out_speed : Real;   // gap proportionality component
      i_part_out_speed : Real;   // gap integral component
      d_part_out_speed : Real;   // gap derivative component
      eff_act_val_speed : Real;   // gap effective process variable
      error_sig_speed : Real;   // gap control deviation
   END_VAR
   VAR CONSTANT
      nc : Real := 0.0;   // "not connected input"
      offs_spd_inc : Real := 0.01;   // 0.01 mm/100ms = 0.1 mm/s
   END_VAR
BEGIN

       //gap control
       //-----------
       //built controller on flag
       //------------------------
       (*
       IF APC.AUTOMATIC THEN
           IF NOT SY.CTL_GAP_SMI THEN  
               SY.CTL_GAP_ON := DC.CTL_GAP_ON;  
           ELSE
               SY.CTL_GAP_ON := FALSE;
           END_IF;
       ELSE
       *)
           //switch on gap control and offset speed control - dia control and melt level tracking must be active
           //---------------------------------------------------------------------------------------------------
           IF (("APC".STATUS = "APC".BODY) AND "SY".CTL_DIA_ON AND "SY".CTL_MLT_LVL_ON) THEN
               //offset speed controller on/off
               //------------------------------
               IF "KYD".CTL_GAP_ON THEN
                   "SY".CTL_OFFS_SPEED_ON  := TRUE;
               ELSIF "KYD".CTL_GAP_OFF THEN
                   "SY".CTL_OFFS_SPEED_ON  := FALSE;
               END_IF;

               //gap control on in automatic when switched on
               //--------------------------------------------
               IF "APC".AUTOMATIC AND NOT "SY".CTL_GAP_SMI THEN
                   "SY".CTL_GAP_ON   :=  "SY".CTL_OFFS_SPEED_ON;
               //gap control off when semi automatic or manual mode is requested
               //---------------------------------------------------------------
               ELSE
                   "SY".CTL_GAP_ON   :=  FALSE;
               END_IF;
           //switch off gap control and offset speed control
           //-----------------------------------------------
           ELSE
               "SY".CTL_GAP_ON           := FALSE;
               "SY".CTL_OFFS_SPEED_ON    := FALSE;
           END_IF;
     //END_IF;

       //set light variable
       //------------------
       "LT".CTL_GAP_ON   :=  "SY".CTL_OFFS_SPEED_ON;   //illuminate gap control button with variable of offset speed control - stays on also in gap semi mode

       //enable of single controller actions
       //----------------------------------- 
       IF ("AC".CTL_GAP_TI > 0.0)   THEN         //i- part
           #int_action_on_gap   :=  true;
       ELSE
           #int_action_on_gap   :=  false;
       END_IF;

       IF ("AC".CTL_GAP_TD > 0.0)   THEN         //d-part
           #der_action_on_gap   :=  true;
       ELSE
           #der_action_on_gap   :=  false;
       END_IF;

       //switch off gap controller
       //-------------------------
       IF NOT "SY".CTL_GAP_ON    THEN 
           #ctl_gap_on  :=  false;
       END_IF;

       //build hand value 
       //----------------
       #hand_gap:= "CM_INSELECT" (auto   := ("APC".AUTOMATIC AND "LT".CTL_GAP_ON AND NOT "SY".CTL_GAP_SMI),        
                               track  := true,
                               ac     := "CTL".SET_GAP_CTL_OFFS,        //The Minus here is to convert the positive Gap Offset into an Decreasement of the Gap.
                                                                      //Positive Gap Offset means that the Drive is moving the Melt level in positiv direction (Up) 
                                                                      //so the Gap is actually going to decrease. This is why a negative Offset is for better understanding because the 
                                                                      //Gap is getting smaller so it should be Minus.              
                               kya    := "KYA".SET_GAP_SMI);     

       //write manual input to zero when controller reset is active or gap control is off 
       //--------------------------------------------------------------------------------
       IF "KYD".GAP_CTRL_RST OR NOT "LT".CTL_GAP_ON THEN
           "KYA".SET_GAP_SMI :=  0.0;
       END_IF;

       //call GAP Standard PID controller
       //--------------------------------
       #GAP_PID(COM_RST         :=  "KYD".GAP_CTRL_RST,                   //restart of controller, resets controller values
               MAN_ON          :=  NOT #ctl_gap_on,                     //switch controller on/off
               PVPER_ON        :=  false,                              //activate reading of peripherie value
               P_SEL           :=  true,                               //proportional action on
               I_SEL           :=  #int_action_on_gap,                  //integral action on
               INT_HOLD        :=  #int_hold_req_gap,                   //integral action hold
               I_ITL_ON        :=  false,                              //initialization of the integral action - set value of I_ITLVAL
               D_SEL           :=  #der_action_on_gap,                  //derivative action on
               CYCLE           :=  T#100ms,                            //sample time
               SP_INT          :=  "DIS".SET_XT_DIA *(-1.0),             //internal setpoint (input polarity changed to negate the output variable)
               PV_IN           :=  "AV".ACT_XT_DIA *(-1.0),              //process variable input (input polarity changed to negate the output variable)
               PV_PER          :=  W#16#0000,                          //process variable peripherial input
               MAN             :=  #hand_gap,                           //hand value   
               GAIN            :=  "AC".CTL_GAP_GN,                      //controller gain
               TI              :=  DINT_TO_TIME(REAL_TO_DINT("AC".CTL_GAP_TI * 1000.0)), //integration time
               TD              :=  DINT_TO_TIME(REAL_TO_DINT("AC".CTL_GAP_TD * 1000.0)), //derivative time
               TM_LAG          :=  DINT_TO_TIME(REAL_TO_DINT("AC".CTL_GAP_T1 * 1000.0)), //time lag of the derivative action
               DEADB_W         :=  0.0,                            //dead band of control deviation
               LMN_HLM         :=  "PAR_MAIN".SET_GAP_OFFS_HL,       //upper limit of controller output as physical value 
               LMN_LLM         :=  "PAR_MAIN".SET_GAP_OFFS_LL,       //lower limit of controller output as physical value
               PV_FAC          :=  1.0,                            //process variable factor (used on peripherial input)
               PV_OFF          :=  0.0,                            //process variable offset
               LMN_FAC         :=  1.0,                            //output standardization(percentage to physical value)
               LMN_OFF         :=  0.0,                            //offset of output value
               I_ITLVAL        :=  0.0,                            //initialization value of the integral action
               DISV            :=  0.0);                           //disturbance variable

               //write output variables of PID controller
               //----------------------------------------
               "CTL".SET_GAP_CTL_OFFS :=  #GAP_PID.LMN;               //controller output variable

               #per_out_gap         :=  #GAP_PID.LMN_PER;            //peripherial controller output variable
               #high_lim_active_gap :=  #GAP_PID.QLMN_HLM;           //high limit of controller output is reached
               #low_lim_active_gap  :=  #GAP_PID.QLMN_LLM;           //low limit of controller output is reached
               #p_part_out_gap      :=  #GAP_PID.LMN_P;              //proportionality component
               #i_part_out_gap      :=  #GAP_PID.LMN_I;              //integral component
               #d_part_out_gap      :=  #GAP_PID.LMN_D;              //derivative component
               #eff_act_val_gap     :=  #GAP_PID.PV;                 //effective process variable 
               #error_sig_gap       :=  #GAP_PID.ER;                 //control deviation  

       //write display values of individual controller parts
       //---------------------------------------------------
       "DIS".GAP_CONT_P:=#p_part_out_gap;
       "DIS".GAP_CONT_D:=#d_part_out_gap;
       "DIS".GAP_CONT_I:=#i_part_out_gap;       

       //write dispaly value of gap controller output
       //--------------------------------------------
       "DIS".SET_GAP_CTL_OFFS := "CTL".SET_GAP_CTL_OFFS;

       //evaluate controller output limits
       //---------------------------------
       IF #high_lim_active_gap OR #low_lim_active_gap   THEN                //check controller limits
           IF (#ctrl_calls_gap > 50) THEN                                   
               IF #high_lim_active_gap AND (#i_part_out_gap > 0.0)   THEN 
                   #int_hold_req_gap    :=  true;                       //set integral action on hold
               ELSIF #low_lim_active_gap AND (#i_part_out_gap < 0.0) THEN 
                   #int_hold_req_gap    :=  true;                       //set integral action on hold
               ELSE 
                   #int_hold_req_gap    :=  false;                      //reset integral action on hold
               END_IF;
           ELSE
               #ctrl_calls_gap  :=  #ctrl_calls_gap + 1;                     //count controller calls
           END_IF;
       ELSE
           #ctrl_calls_gap      :=  0;                                  //reset controller call counts
           #int_hold_req_gap    :=  false;                              //reset integral action hold request
       END_IF; 

       //switch on gap controller
       //------------------------
       IF "SY".CTL_GAP_ON    THEN 
           #ctl_gap_on  :=  true;
       END_IF;

       //offset speed control
       //--------------------
       //Calculate Melt gap offset from set point of speed offset - FB called on 100ms interrupt
       //---------------------------------------------------------------------------------------
       IF "SY".CTL_OFFS_SPEED_ON THEN
           "DIS".ACT_MLT_GAP_OFFS:= "DIS".ACT_MLT_GAP_OFFS + "CTL".SET_SPEED_OFFS * (-1.0) / 600.0;
       ELSE
           "DIS".ACT_MLT_GAP_OFFS:= 0.0;
       END_IF;

       //switch off offset speed controller
       //----------------------------------
       IF NOT "SY".CTL_OFFS_SPEED_ON THEN 
           #ctl_offs_spd_on  :=  false;
           //ramp controller output to zero, when offset speed control is switched off
           //-------------------------------------------------------------------------
           IF ("CTL".SET_SPEED_OFFS > 0.0) THEN      //positive set point active
               #hand_offs_spd   := "CTL".SET_SPEED_OFFS - #offs_spd_inc;
               IF (#hand_offs_spd < 0.0) THEN
                   #hand_offs_spd    :=  0.0;
               END_IF;
           ELSE
               IF ("CTL".SET_SPEED_OFFS < 0.0) THEN  //negative set point active
                   #hand_offs_spd    := "CTL".SET_SPEED_OFFS + #offs_spd_inc;
                   IF (#hand_offs_spd > 0.0) THEN
                       #hand_offs_spd    :=  0.0;
                   END_IF;
               ELSE
                   #hand_offs_spd    :=  0.0;
               END_IF;
           END_IF;
       END_IF;

       //enable of single controller actions
       //----------------------------------- 
       IF ("AC".CTL_OFFS_SPEED_TI > 0.0)   THEN         //i- part
           #int_action_on_speed   :=  true;
       ELSE
           #int_action_on_speed   :=  false;
       END_IF;

       IF ("AC".CTL_OFFS_SPEED_TD > 0.0)   THEN         //d-part
           #der_action_on_speed   :=  true;
       ELSE
           #der_action_on_speed   :=  false;
       END_IF;

       //call Offset Speed Standard PID controller
       //--------------------------------
       #OFFS_SPEED_PID(COM_RST  :=  "KYD".GAP_CTRL_RST,                   //restart of controller, resets controller values
               MAN_ON          :=  NOT #ctl_offs_spd_on,                //switch controller on/off
               PVPER_ON        :=  false,                              //activate reading of peripherie value
               P_SEL           :=  true,                               //proportional action on
               I_SEL           :=  #int_action_on_speed,                //integral action on
               INT_HOLD        :=  #int_hold_req_speed,                 //integral action hold
               I_ITL_ON        :=  false,                              //initialization of the integral action - set value of I_ITLVAL
               D_SEL           :=  #der_action_on_speed,                //derivative action on
               CYCLE           :=  T#100ms,                            //sample time
               SP_INT          :=  "CTL".SET_GAP_CTL_OFFS * (-1.0),      //internal setpoint (input polarity changed to negate the output variable)
               PV_IN           :=  "DIS".ACT_MLT_GAP_OFFS * (-1.0),      //process variable input (input polarity changed to negate the output variable)
               PV_PER          :=  W#16#0000,                          //process variable peripherial input
               MAN             :=  #hand_offs_spd,                      //hand value as percentaged input
               GAIN            :=  "AC".CTL_OFFS_SPEED_GN,               //controller gain
               TI              :=  DINT_TO_TIME(REAL_TO_DINT("AC".CTL_OFFS_SPEED_TI * 1000.0)), //integration time
               TD              :=  DINT_TO_TIME(REAL_TO_DINT("AC".CTL_OFFS_SPEED_TD * 1000.0)), //derivative time
               TM_LAG          :=  DINT_TO_TIME(REAL_TO_DINT("AC".CTL_OFFS_SPEED_T1 * 1000.0)), //time lag of the derivative action
               DEADB_W         :=  0.0,                                //dead band of control deviation
               LMN_HLM         :=  "PAR_MAIN".SET_OFFS_SPEED_HL,         //upper limit of controller output as percentaged value 
               LMN_LLM         :=  "PAR_MAIN".SET_OFFS_SPEED_LL,         //lower limit of controller output as percentaged value
               PV_FAC          :=  1.0,                                //process variable factor (used on peripherial input)
               PV_OFF          :=  0.0,                                //process variable offset
               LMN_FAC         :=  1.0,                                //output standardization(percentage to physical value)
               LMN_OFF         :=  0.0,                                //offset of output value
               I_ITLVAL        :=  0.0,                                //initialization value of the integral action
               DISV            :=  0.0);                               //disturbance variable

               //write output variables of PID controller
               //----------------------------------------
               "CTL".SET_SPEED_OFFS:=  #OFFS_SPEED_PID.LMN;           //controller output variable as physical value

               #per_out_speed         :=  #OFFS_SPEED_PID.LMN_PER;       //peripherial controller output variable
               #high_lim_active_speed :=  #OFFS_SPEED_PID.QLMN_HLM;      //high limit of controller output is reached
               #low_lim_active_speed  :=  #OFFS_SPEED_PID.QLMN_LLM;      //low limit of controller output is reached
               #p_part_out_speed      :=  #OFFS_SPEED_PID.LMN_P;         //proportionality component
               #i_part_out_speed      :=  #OFFS_SPEED_PID.LMN_I;         //integral component
               #d_part_out_speed      :=  #OFFS_SPEED_PID.LMN_D;         //derivative component
               #eff_act_val_speed     :=  #OFFS_SPEED_PID.PV;            //effective process variable 
               #error_sig_speed       :=  #OFFS_SPEED_PID.ER;            //control deviation  

       //write display values of individual controller parts
       //---------------------------------------------------
       "DIS".OFFS_SPD_CONT_P:=#p_part_out_speed;
       "DIS".OFFS_SPD_CONT_D:=#d_part_out_speed;
       "DIS".OFFS_SPD_CONT_I:=#i_part_out_speed;          

       //write dispaly value of offset speed controller output
       //-----------------------------------------------------
       "DIS".SET_SPEED_OFFS:=    "CTL".SET_SPEED_OFFS; 

       //evaluate controller output limits
       //---------------------------------
       IF #high_lim_active_speed OR #low_lim_active_speed   THEN                //check controller limits
           IF (#ctrl_calls_speed > 50) THEN                                   
               IF #high_lim_active_speed AND (#i_part_out_speed > 0.0)   THEN 
                   #int_hold_req_speed    :=  true;                       //set integral action on hold
               ELSIF #low_lim_active_speed AND (#i_part_out_speed < 0.0) THEN 
                   #int_hold_req_speed    :=  true;                       //set integral action on hold
               ELSE 
                   #int_hold_req_speed    :=  false;                      //reset integral action on hold
               END_IF;
           ELSE
               #ctrl_calls_speed  :=  #ctrl_calls_speed + 1;                     //count controller calls
           END_IF;
       ELSE
           #ctrl_calls_speed      :=  0;                                  //reset controller call counts
           #int_hold_req_speed    :=  false;                              //reset integral action hold request
       END_IF;

       //switch on offset speed controller
       //---------------------------------
       IF "SY".CTL_OFFS_SPEED_ON THEN 
           #ctl_offs_spd_on  :=  true;
       END_IF;
END_FUNCTION_BLOCK

FUNCTION_BLOCK "CM_SEL_CTRL_ALG"   // FB146, SCL
{ S7_Optimized_Access := 'FALSE' }
VERSION : 0.0
// --------------------------------------------------------------------------------
//     program     :    CM_SEL_CTRL_ALG
//     description :    do selection of PID control algorithm    
//     name        :    G. Eibelsh鋟ser
//     date        :    19.09.2007
// 
//     revision    :
//     name        :
//     date        :    
//                     (c)CGS
//     --------------------------------------------------------------------------------
   VAR
      prs_ctrl_std_alg : Real;
      dia_ctrl_std_alg : Real;
      htr_1_ctrl_std_alg : Real;
      spd_ctrl_std_alg : Real;
      cruc_rot_ctrl_std_alg : Real;
      mlt_tmp_ctrl_std_alg : Real;
      grw_rte_ctrl_std_alg : Real;
   END_VAR
BEGIN


       //set all loops to Siemens standard algorithm (Cont_C)
       //----------------------------------------------------
       "PAR_MAIN".PRS_CTRL_STD_ALG           :=  1.0;    
       "PAR_MAIN".DIA_CTRL_STD_ALG           :=  1.0;
       "PAR_MAIN".HTR_1_CTRL_STD_ALG         :=  1.0;
       "PAR_MAIN".SPD_CTRL_STD_ALG           :=  1.0;
       "PAR_MAIN".CRUC_ROT_CTRL_STD_ALG      :=  1.0;
       "PAR_MAIN".MLT_TMP_CTRL_STD_ALG       :=  1.0;
       "PAR_MAIN".GRW_RTE_CTRL_STD_ALG       :=  1.0;    

       //selection of pressure control algorithm
       //---------------------------------------
       IF NOT "LT".CTL_PRS_ON THEN                               //control loop is off  
           //set algorithm flag 
           //------------------
           IF (REAL_TO_INT("PAR_MAIN".PRS_CTRL_STD_ALG) = 1)    THEN
               "DV".PRS_CTRL_STD_ALG :=  TRUE;                   //standard Siemens algorithm
           ELSE
               "DV".PRS_CTRL_STD_ALG :=  FALSE;                  //CGS modified algorithm
           END_IF;

           #prs_ctrl_std_alg    :=  "PAR_MAIN".PRS_CTRL_STD_ALG;  //store actual selection while loop is off  

       ELSE                                                    //control loop is on
           "PAR_MAIN".PRS_CTRL_STD_ALG   :=  #prs_ctrl_std_alg;   //overwrite section parameter
       END_IF;       

       //selection of diameter control algorithm
       //---------------------------------------
       IF NOT "LT".CTL_DIA_ON THEN                               //control loop is off  
           //set algorithm flag 
           //------------------
           IF (REAL_TO_INT("PAR_MAIN".DIA_CTRL_STD_ALG) = 1)    THEN
               "DV".DIA_CTRL_STD_ALG :=  TRUE;                   //standard Siemens algorithm
           ELSE
               "DV".DIA_CTRL_STD_ALG :=  FALSE;                  //CGS modified algorithm
           END_IF;

           #dia_ctrl_std_alg    :=  "PAR_MAIN".DIA_CTRL_STD_ALG;  //store actual selection while loop is off  

       ELSE                                                    //control loop is on
           "PAR_MAIN".DIA_CTRL_STD_ALG   :=  #dia_ctrl_std_alg;   //overwrite section parameter
       END_IF;       

       //selection of heater temperature control algorithm
       //-------------------------------------------------
       IF NOT "LT".CTL_HTR_1_TMP_ON THEN                             //control loop is off  
           //set algorithm flag 
           //------------------
           IF (REAL_TO_INT("PAR_MAIN".HTR_1_CTRL_STD_ALG) = 1)    THEN
               "DV".HTR_1_CTRL_STD_ALG :=  TRUE;                     //standard Siemens algorithm
           ELSE
               "DV".HTR_1_CTRL_STD_ALG :=  FALSE;                    //CGS modified algorithm
           END_IF;

           #htr_1_ctrl_std_alg    :=  "PAR_MAIN".HTR_1_CTRL_STD_ALG;  //store actual selection while loop is off  

       ELSE                                                        //control loop is on
           "PAR_MAIN".HTR_1_CTRL_STD_ALG   :=  #htr_1_ctrl_std_alg;   //overwrite section parameter
       END_IF;       

       //selection of average speed control algorithm
       //--------------------------------------------
       IF NOT "LT".CTL_AV_SPD_ON THEN                             //control loop is off  
           //set algorithm flag 
           //------------------
           IF (REAL_TO_INT("PAR_MAIN".SPD_CTRL_STD_ALG) = 1)    THEN
               "DV".SPD_CTRL_STD_ALG :=  TRUE;                     //standard Siemens algorithm
           ELSE
               "DV".SPD_CTRL_STD_ALG :=  FALSE;                    //CGS modified algorithm
           END_IF;

           #spd_ctrl_std_alg    :=  "PAR_MAIN".SPD_CTRL_STD_ALG;      //store actual selection while loop is off  

       ELSE                                                        //control loop is on
           "PAR_MAIN".SPD_CTRL_STD_ALG   :=  #spd_ctrl_std_alg;   //overwrite section parameter
       END_IF;       

       //selection of average crucible rotation control algorithm
       //--------------------------------------------------------
       IF NOT "LT".CTL_AV_CRUC_ROT_ON THEN                                   //control loop is off  
           //set algorithm flag 
           //------------------
           IF (REAL_TO_INT("PAR_MAIN".CRUC_ROT_CTRL_STD_ALG) = 1)    THEN
               "DV".CRUC_ROT_CTRL_STD_ALG    :=  TRUE;                       //standard Siemens algorithm
           ELSE
               "DV".CRUC_ROT_CTRL_STD_ALG    :=  FALSE;                      //CGS modified algorithm
           END_IF;

           #cruc_rot_ctrl_std_alg    :=  "PAR_MAIN".CRUC_ROT_CTRL_STD_ALG   ;  //store actual selection while loop is off  

       ELSE                                                                //control loop is on
           "PAR_MAIN".CRUC_ROT_CTRL_STD_ALG      :=  #cruc_rot_ctrl_std_alg;   //overwrite section parameter
       END_IF;       

       //selection of melt temperature control algorithm
       //-----------------------------------------------
       IF NOT "LT".CTL_MELT_TMP_1_ON THEN                                   //control loop is off  
           //set algorithm flag 
           //------------------
           IF (REAL_TO_INT("PAR_MAIN".MLT_TMP_CTRL_STD_ALG) = 1)    THEN
               "DV".MLT_TMP_CTRL_STD_ALG    :=  TRUE;                        //standard Siemens algorithm
           ELSE
               "DV".MLT_TMP_CTRL_STD_ALG    :=  FALSE;                       //CGS modified algorithm
           END_IF;

           #mlt_tmp_ctrl_std_alg    :=  "PAR_MAIN".MLT_TMP_CTRL_STD_ALG;      //store actual selection while loop is off  

       ELSE                                                                //control loop is on
           "PAR_MAIN".MLT_TMP_CTRL_STD_ALG   :=  #mlt_tmp_ctrl_std_alg;       //overwrite section parameter
       END_IF;       

       //selection of growth control algorithm
       //-------------------------------------
       IF NOT "LT".CTL_GRO_ON THEN                                           //control loop is off  
           //set algorithm flag 
           //------------------
           IF (REAL_TO_INT("PAR_MAIN".GRW_RTE_CTRL_STD_ALG) = 1)    THEN
               "DV".GRW_RTE_CTRL_STD_ALG    :=  TRUE;                        //standard Siemens algorithm
           ELSE
               "DV".GRW_RTE_CTRL_STD_ALG    :=  FALSE;                       //CGS modified algorithm
           END_IF;

           #grw_rte_ctrl_std_alg    :=  "PAR_MAIN".GRW_RTE_CTRL_STD_ALG;      //store actual selection while loop is off  

       ELSE                                                                //control loop is on
           "PAR_MAIN".GRW_RTE_CTRL_STD_ALG   :=  #grw_rte_ctrl_std_alg;        //overwrite section parameter
       END_IF;
END_FUNCTION_BLOCK

FUNCTION_BLOCK "CM_SLD_AVG"   // FB147, SCL
{ S7_Optimized_Access := 'FALSE' }
VERSION : 0.0
// --------------------------------------------------------------------------------
//     program     :    CM_SLD_AVG
//     description :    calculation of sliding average
//     name        :    G. Eibelsh鋟ser
//     date        :    31.01.2007
// 
//     revision    :  
//     name        :   
//     date        :    
// 
//                     (c)CGS
//     --------------------------------------------------------------------------------
   VAR_INPUT
      calc_on : Bool;   // calculation activated
      order : Int;   // order of sliding average
      u_in : Real;   // input value
      ts_in : Real;   // sample time
      tc_in : Real;   // call time
   END_VAR
   VAR_IN_OUT
      y_out : Real;   // output value
   END_VAR
   VAR
      data_rec_init : Bool;   // data record initialisation
      calc_cycle : Int;   // calculation cycle
      i : Int;   // record index
      amt_of_val : Int;   // amount of valid values in data record
      order_old : Int;   // actual order of sliding average
      record_sum : Real;   // summation of record data
      data_rec : Array[1..300] of Real;   // data record
   END_VAR
BEGIN


       IF #calc_on  THEN        //caculation enabled
           IF #calc_cycle >= REAL_TO_INT(#ts_in / #tc_in)   THEN 
               #calc_cycle  :=  1;

               IF (#order > 300)    THEN
                   #order   :=  300;        //limit order to a maximum of 300
               END_IF;

               IF (#order > 0)  THEN 

                   //check if order has changed
                   //--------------------------
                   IF (#order <> #order_old) THEN
                       #data_rec_init   :=  true;
                       #record_sum      :=  0.0;   //reset record sum
                       #i               :=  0; 
                   END_IF;

                   //increment record index each call
                   //--------------------------------
                   #i   :=  #i + 1;

                   //deduct oldest value from record sum
                   //-----------------------------------
                   IF NOT #data_rec_init    THEN    //record initialisation done
                       #record_sum  :=  #record_sum - #data_rec[#i];
                   END_IF;

                   //store new input value in record
                   //-------------------------------
                   #data_rec[#i] :=  #u_in;

                   //add newest value to record sum
                   //------------------------------
                   #record_sum  :=  #record_sum + #data_rec[#i];

                   //read amount of valid values in data record
                   //------------------------------------------
                   IF #data_rec_init THEN 
                       #amt_of_val  :=  #i;
                   ELSE
                       #amt_of_val  :=  #order;
                   END_IF;

                   //calculate average value
                   //-----------------------
                   #y_out   :=  #record_sum  / #amt_of_val;

                   //reset record index when maximum amount of values is reached
                   //-----------------------------------------------------------
                   IF (#i >= #order)  THEN
                       #i               :=  0;
                       #data_rec_init   :=  FALSE;
                   END_IF;

                   //store order setting
                   //-------------------
                   #order_old   :=  #order;  

               ELSE         
                   //no average calculation - input = output
                   //---------------------------------------
                   #y_out   :=  #u_in;       
               END_IF;
           ELSE 
               #calc_cycle  :=  #calc_cycle + 1;
           END_IF;

       //caculation disabled - reset variables and flags
       //-----------------------------------------------
       ELSE                
           #i               :=  0;
           #calc_cycle      :=  1;
           #record_sum      :=  0.0;
           #y_out           :=  0.0;
           #data_rec_init   :=  TRUE;

       END_IF;
END_FUNCTION_BLOCK

